RoboDK station: ex1.rdk

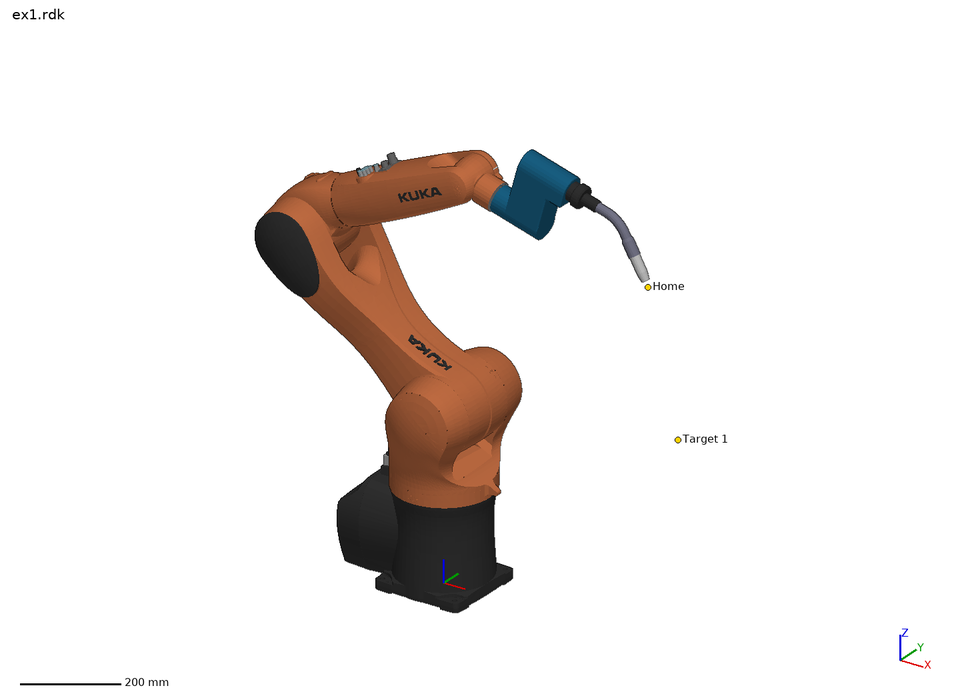
[picture v0: the station drawn from its stored meshes, robots at their saved joint values, targets as dots, program paths as lines]
Station Offline programming - Weld test KUKA. Poses are relative to the parent item; angles as X-Y-Z fixed-axis rotations.
  - frame KUKA KR 6 R900 sixx Base at (0, 0, 0) mm
    - robot KUKA KR 6 R900 sixx: 6 axes, payload 6 kg, reach 901 mm, repeatability 0.03 mm, weight 52 kg
        modified DH rows (alpha deg, a mm, theta deg, d mm): 0, 0, 0, 400; -90, 25, 0, 0; 0, 455, -90, 0; -90, 35, 0, 420; 90, 0, 0, 0; -90, 0, 180, 80
        joint limits [-170, -190, -120, -185, -120, -350] to [170, 45, 156, 185, 120, 350]; home [0, -90, 90, 0, 0, 0]; saved at [0, -138.016, 114.252, 0, 39.328, 0]
      - tool Weld gun, TCP at (-4, 0, 371.3) mm, rotated rx 0 ry 45 rz 0 deg, size 299.9 x 60 x 318.3 mm
    - target Home (Cartesian target) at (492.9, 0, 788.4) mm, rotated rx -180 ry 29.44 rz -180 deg; joints [0, -138.016, 114.252, 0, 39.328, 0] of KUKA KR 6 R900 sixx
    - target Target 1 (Cartesian target) at (564.87, 0, 471.83) mm, rotated rx -180 ry 0 rz -180 deg; joints [0, -116.511, 123.863, 0, 37.648, 0] of KUKA KR 6 R900 sixx
  - Python program Hexagonal path (listed below)

--- Python program Hexagonal path ---
from robolink import *    # API to communicate with RoboDK
from robodk import *      # robodk robotics toolbox

# Any interaction with RoboDK must be done through RDK:
RDK = Robolink()

# get the robot by name:
robot = RDK.Item('', ITEM_TYPE_ROBOT)

# get the home target and the welding targets:
home = RDK.Item('Home')
target = RDK.Item('Target 1')

# get the pose of the target (4x4 matrix representing position and orientation):
poseref = target.Pose()

# move the robot to home, then to the Target 1:
robot.MoveJ(home)
robot.MoveJ(target)

# make an hexagon around the Target 1:
for i in range(7):
    ang = i*2*pi/6 #angle: 0, 60, 120, ...
    posei = poseref*rotz(ang)*transl(200,0,0)*rotz(-ang)
    robot.MoveL(posei)

# move back to the center, then home:
robot.MoveL(target)
robot.MoveJ(home)
